{attribute 'global_init_slot' := '40500'} //https://infosys.beckhoff.com/index.php?content=../content/1031/tc3_plc_intro/2529649291.html&id=
VAR_GLOBAL CONSTANT
	MaxNrofMessages: UINT:= 30;
	emptySkill : FB_1_Skill; //emptySkill
END_VAR


{attribute 'global_init_slot' := '40600'} //https://infosys.beckhoff.com/index.php?content=../content/1031/tc3_plc_intro/2529649291.html&id=
//Skills
VAR_GLOBAL
	TS_Count: Skill_Counter;
	TS_3P: TEST_Skill_3Points;
	TS_2P: TEST_Skill_2Points;
	TS_varP: TEST_Skill_varP;

END_VAR



{attribute 'global_init_slot' := '40700'} //https://infosys.beckhoff.com/index.php?content=../content/1031/tc3_plc_intro/2529649291.html&id=
//Robots
VAR_GLOBAL


	T_UR: ROBOT_UR :=(
		Skills:= [ADR(TS_Count),ADR(TS_3P),ADR(TS_2P),ADR(TS_varP)]
	);
	

END_VAR


VAR_GLOBAL

END_VAR

(* stored: Version 1.1.0.1, ProductVersion 3.1.4026.18
   GVL TESTSETUP: Id {afb3172e-52f3-48ee-939b-708551773a13} *)
